ADAPTER AB2 (* bidirectional Adapter Interface for 1 Event and 1 Byte *)
  (* Standard: 61499-1; Description: Copyright (c) 2025 HR Agrartechnik GmbH This program and the accompanying materials are made available under the terms of the Eclipse Public License 2.0 which is available at https://www.eclipse.org/legal/epl-2.0/ SPDX-License-Identifier: EPL-2.0 *)
  (* Version 1.0, 2025-01-24, Franz Höpfinger, HR Agrartechnik GmbH, Initial Version *)
  PACKAGE adapter::types::bidirectional;
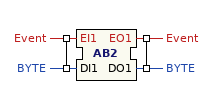
  EVENT_INPUT
    EI1 WITH DI1; (* Request (or Indication) *)
  END_EVENT
  EVENT_OUTPUT
    EO1 WITH DO1; (* Indication (or Request) *)
  END_EVENT
  VAR_INPUT
    DI1 : BYTE; (* Request (or Indication) to Socket *)
  END_VAR
  VAR_OUTPUT
    DO1 : BYTE; (* Indication (or Request) Data from Plug *)
  END_VAR
END_ADAPTER
